(* IEC 61131-3 sources: Edge_Computing_on_PLC/st_app_with_rust_lib/PROGRAM/POU_FULL_ST, 1 file *)

(* ---- main.st ---- *)
PROGRAM ST_PRG_WITH_RS_LIB
    VAR
        // Rust high-efficiency computing lib input
        // temperature_data:   ARRAY[0..49] OF REAL;
        // pressure_data:      ARRAY[0..49] OF REAL;
        // humidity_data:      ARRAY[0..49] OF REAL;

        // Rust high-efficiency computing lib output
        t_mean:                 REAL;
        t_variance:             REAL;
        t_std_deviation:        REAL;
        t_z_score:              REAL;
        p_mean:                 REAL;
        p_variance:             REAL;
        p_std_deviation:        REAL;
        p_z_score:              REAL;
        h_mean:                 REAL;
        h_variance:             REAL;
        h_std_deviation:        REAL;
        h_z_score:              REAL;

        // Rust spectrum estimation lib output
        t_freq:                 REAL;
        t_ampl:                 REAL;
        t_offset:               REAL;
        t_phase:                REAL;
        p_freq:                 REAL;
        p_ampl:                 REAL;
        p_offset:               REAL;
        p_phase:                REAL;
        h_freq:                 REAL;
        h_ampl:                 REAL;
        h_offset:               REAL;
        h_phase:                REAL;

        // Rust high-efficiency computing lib
        zad:                    z_anm_detc;

        // Rust spectrum estimation lib output
        sa:                     spctrm_anlys;

        // Counter
        // counter:            INT := 0;

        // Anomaly Flag
        t_anm_flag:             BOOL := FALSE;
        p_anm_flag:             BOOL := FALSE;
        h_anm_flag:             BOOL := FALSE;

    END_VAR

    // Update data for each cycle
    zad(
        temperature := temperature / 100.0,
        pressure := pressure / 100.0,
        humidity := humidity / 100.0,
        t_mean => t_mean,
        t_variance => t_variance,
        t_standard_deviation => t_std_deviation,
        t_z_score => t_z_score,
        p_mean => p_mean,
        p_variance => p_variance,
        p_standard_deviation => p_std_deviation,
        p_z_score => p_z_score,
        h_mean => h_mean,
        h_variance => h_variance,
        h_standard_deviation => h_std_deviation,
        h_z_score => h_z_score
    );

    sa(
        temperature := temperature / 100.0,
        humidity := humidity / 100.0,
        pressure := pressure / 100.0,
        t_freq => t_freq,
        t_ampl => t_ampl,
        t_offset => t_offset,
        t_phase => t_phase,
        h_freq => h_freq,
        h_ampl => h_ampl,
        h_offset => h_offset,
        h_phase => h_phase,
        p_freq => p_freq,
        p_ampl => p_ampl,
        p_offset => p_offset,
        p_phase => p_phase
    );

    // Check whether temperature's Z score has anomaly.
    IF t_z_score >= 1.5 THEN
        t_anm_flag := TRUE;
    ELSIF t_z_score <= -1.5 THEN
        t_anm_flag := TRUE;
    ELSE
        t_anm_flag := FALSE;
    END_IF

    // Check whether pressure's Z score has anomaly.
    IF p_z_score >= 1.5 THEN
        p_anm_flag := TRUE;
    ELSIF p_z_score <= -1.5 THEN
        p_anm_flag := TRUE;
    ELSE
        p_anm_flag := FALSE;
    END_IF

    // Check whether humidity's Z score has anomaly.
    IF h_z_score >= 1.5 THEN
        h_anm_flag := TRUE;
    ELSIF h_z_score <= -1.5 THEN
        h_anm_flag := TRUE;
    ELSE
        h_anm_flag := FALSE;
    END_IF

END_PROGRAM
